FUNCTION_BLOCK Test_LTrimEx_HandlesEmptySubject EXTENDS T_UnitTestBase
VAR_INPUT
END_VAR
VAR_OUTPUT
END_VAR
VAR
    SubjectString : T_MaxString := '';
END_VAR

{attribute 'analysis' := '-33'} // inhibit unused variable warning
METHOD RunTest
IF Retest THEN
	SUPER^.Init();
END_IF

IF TestCompleted THEN
	RETURN;
END_IF

AssertEquals_STRING(Expected := '',
                    Actual   := F_LTrimEx(n := 1, str := SubjectString),
                    Message  := 'F_LTrimEx(SubjectString)');

TestCompleted := TRUE;
END_METHOD

END_FUNCTION_BLOCK

(* stored: Version 1.1.0.1, ProductVersion 3.1.4024.12
   POU Test_LTrimEx_HandlesEmptySubject: Id {702686f4-9c00-0487-3922-1333a8a31a5e}, SpecialFunc None
   Method RunTest: Id {7ab67b22-70fa-03c2-2661-d7b149df0097} *)
